PROGRAM MAIN
VAR
	cluster_control : FB_Cluster_Control();
	sita_out : REAL;
	sita_in1 : REAL;
	sita_in2 : REAL;
	sita_setout : FB_SetOutput();
END_VAR

cluster_control();

//sita_out := F_SetOutput_LatestInput(in1 := TO_REAL(sita_in1),in2 := TO_REAL(sita_in2));


sita_setout(io_in1 := sita_in1,io_in2 := sita_in2, o_set_value => sita_out);

END_PROGRAM

(* stored: Version 1.1.0.1, ProductVersion 3.1.4024.12
   POU MAIN: Id {cc4f0746-d0f9-4454-8a3d-2c3137eb714f}, SpecialFunc None *)
